(* PLC project Blank Project, Blank Blank 1.0 *)
(* stored: creationDateTime 2016-05-18T21:14:07, modificationDateTime 2020-06-30T11:51:56 *)

FUNCTION_BLOCK close_angle
  VAR_INPUT
    current_ang1 : INT;
    current_ang2 : INT;
    ang1 : INT;
    ang2 : INT;
  END_VAR
  VAR
    window : INT := 1;
  END_VAR
  VAR_OUTPUT
    boolean : BOOL := false;
  END_VAR

            IF (current_ang1 >= (ang1 - window)) AND (current_ang1 <= (ang1 + window)) THEN
  IF (current_ang2 >= (ang2 - window)) AND (current_ang2 <= (ang2 + window)) THEN
    boolean := true;
  ELSE
    boolean := false;
  END_IF;
ELSE
  boolean := false;
END_IF;
          
END_FUNCTION_BLOCK

PROGRAM My_Program
  VAR
    Tau1 AT %IW0 : INT;
    Tau2 AT %IW1 : INT;
    Theta1 AT %IW2 : INT;
    Theta2 AT %IW3 : INT;
    Theta1_out AT %QW0 : INT;
    Theta2_out AT %QW1 : INT;
    Theta1_sp AT %QW2 : INT;
    Theta2_sp AT %QW3 : INT;
    Length1 AT %QW4 : UINT := 100;
    Length2 AT %QW5 : UINT := 50;
    count AT %QW6 : INT := 0;
    auto_start1 AT %QW7 : INT := 10;
    auto_start2 AT %QW8 : INT := 20;
    auto_end1 AT %QW9 : INT := 20;
    auto_end2 AT %QW10 : INT := 30;
    completed AT %QW11 : INT := 0;
    remaining AT %QW12 : INT := 0;
    mode AT %QX0.0 : BOOL := 0;
    start AT %QX0.1 : BOOL := 0;
    oscillator AT %QX0.2 : BOOL := 0;
    switch AT %QX0.3 : BOOL := 0;
  END_VAR
  VAR
    CTU0 : CTU;
    TP0 : TP;
    close_angle0 : close_angle;
    close_angle1 : close_angle;
    TON0 : TON;
    TON1 : TON;
  END_VAR
  VAR  (* added by the conversion: wires and edge detectors of the diagram *)
    R_TRIG1 : R_TRIG;
    F_TRIG2 : F_TRIG;
    R_TRIG3 : R_TRIG;
    _MUL76_OUT : INT;
    _MOD28_ENO : BOOL;
    _MOD28_OUT : INT;
    _NOT44_OUT : BOOL;
    _MOVE42_ENO : BOOL;
    _MOVE42_OUT : INT;
  END_VAR

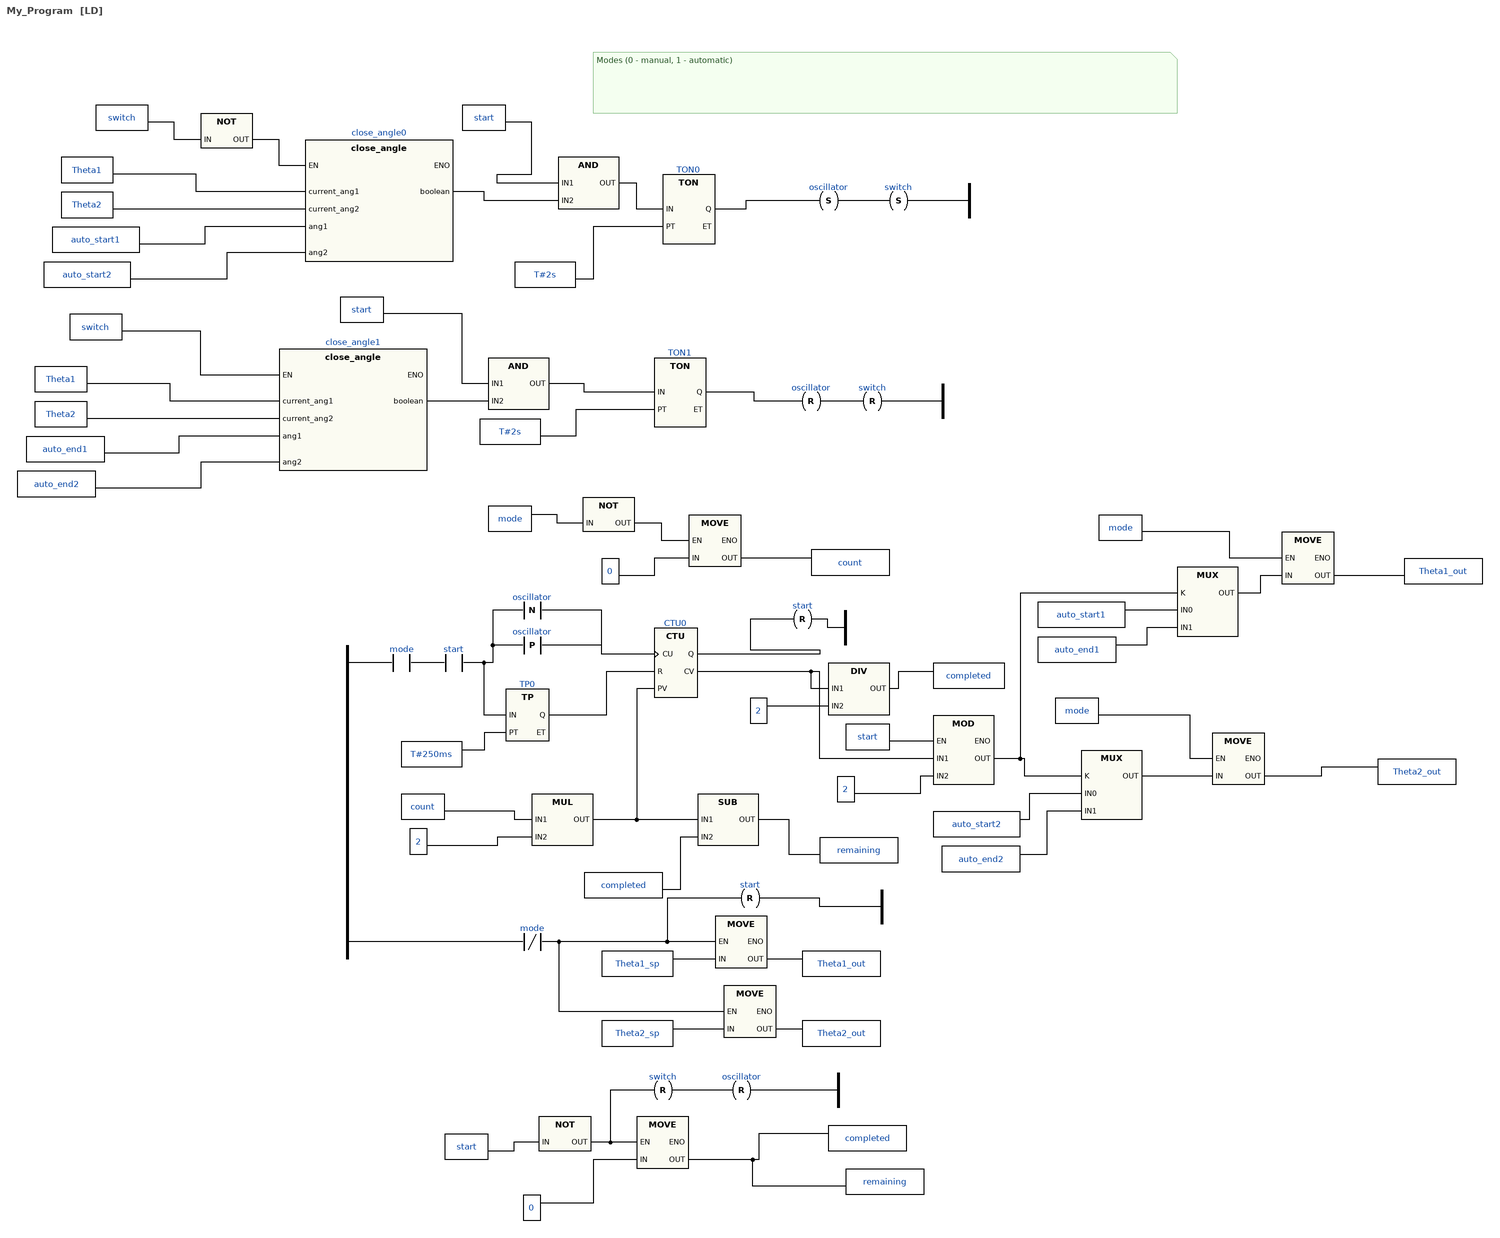
(* LD diagram, written out as Structured Text *)
(* Modes (0 - manual, 1 - automatic) *)
close_angle0(EN := NOT switch, current_ang1 := Theta1, current_ang2 := Theta2, ang1 := auto_start1, ang2 := auto_start2);
TON0(IN := start AND close_angle0.boolean, PT := T#2s);
IF TON0.Q THEN oscillator := TRUE; END_IF;
IF TON0.Q THEN switch := TRUE; END_IF;
close_angle1(EN := switch, current_ang1 := Theta1, current_ang2 := Theta2, ang1 := auto_end1, ang2 := auto_end2);
TON1(IN := start AND close_angle1.boolean, PT := T#2s);
IF TON1.Q THEN oscillator := FALSE; END_IF;
IF TON1.Q THEN switch := FALSE; END_IF;
IF NOT mode THEN count := 0; END_IF;
R_TRIG1(CLK := oscillator);
F_TRIG2(CLK := oscillator);
R_TRIG3(CLK := mode AND start AND (R_TRIG1.Q OR F_TRIG2.Q));
TP0(IN := mode AND start, PT := T#250ms);
_MUL76_OUT := count * 2;
CTU0(CU := R_TRIG3.Q, R := TP0.Q, PV := _MUL76_OUT);
_MOD28_OUT := MOD(EN := start, IN1 := CTU0.CV, IN2 := 2, ENO => _MOD28_ENO);
IF mode THEN Theta1_out := MUX(_MOD28_OUT, auto_start1, auto_end1); END_IF;
IF CTU0.Q THEN start := FALSE; END_IF;
completed := CTU0.CV / 2;
IF mode THEN Theta2_out := MUX(_MOD28_OUT, auto_start2, auto_end2); END_IF;
remaining := _MUL76_OUT - completed;
IF NOT mode THEN start := FALSE; END_IF;
IF NOT mode THEN Theta1_out := Theta1_sp; END_IF;
IF NOT mode THEN Theta2_out := Theta2_sp; END_IF;
_NOT44_OUT := NOT start;
IF _NOT44_OUT THEN switch := FALSE; END_IF;
IF _NOT44_OUT THEN oscillator := FALSE; END_IF;
_MOVE42_OUT := MOVE(EN := _NOT44_OUT, IN := 0, ENO => _MOVE42_ENO);
IF _MOVE42_ENO THEN completed := _MOVE42_OUT; END_IF;
IF _MOVE42_ENO THEN remaining := _MOVE42_OUT; END_IF;
END_PROGRAM

CONFIGURATION Config0
  RESOURCE Res0 ON PLC
    TASK TaskMain(INTERVAL := T#50ms, PRIORITY := 0);
    PROGRAM Inst0 WITH TaskMain : My_Program;
  END_RESOURCE
END_CONFIGURATION
